LIN {X 0,Y 150.243,Z 1030.549,A -85,B 0,C 180,E1 -31632.284,E2 -31632.284} C_VEL
LIN {X 0,Y 145.871,Z 1032.288,A -85,B 0,C 180,E1 -31632.248,E2 -31632.248} C_VEL
LIN {X 0,Y 142.516,Z 1033.901,A -85,B 0,C 180,E1 -31631.848,E2 -31631.848} C_VEL
LIN {X 0,Y 134.858,Z 1038.027,A -85,B 0,C 180,E1 -31630.012,E2 -31630.012} C_VEL
LIN {X 0,Y 127.872,Z 1041.883,A -85,B 0,C 180,E1 -31627.541,E2 -31627.541} C_VEL
LIN {X 0,Y 116.114,Z 1047.754,A -85,B 0,C 180,E1 -31622.075,E2 -31622.075} C_VEL
LIN {X 0,Y 107.865,Z 1051.272,A -85,B 0,C 180,E1 -31617.134,E2 -31617.134} C_VEL
LIN {X 0,Y 99.707,Z 1054.249,A -85,B 0,C 180,E1 -31610.636,E2 -31610.636} C_VEL
LIN {X 0,Y 93.129,Z 1056.253,A -85,B 0,C 180,E1 -31603.085,E2 -31603.085} C_VEL
LIN {X 0,Y 88.672,Z 1057.261,A -85,B 0,C 180,E1 -31594.546,E2 -31594.546} C_VEL
LIN {X 0,Y 87.304,Z 1057.479,A -85,B 0,C 180,E1 -31590,E2 -31590} C_VEL
LIN {X 0,Y 90.603,Z 1056.917,A -85,B 0,C 180,E1 -31581.075,E2 -31581.075} C_VEL
LIN {X 0,Y 96.175,Z 1055.425,A -85,B 0,C 180,E1 -31573.005,E2 -31573.005} C_VEL
LIN {X 0,Y 103.623,Z 1052.922,A -85,B 0,C 180,E1 -31565.988,E2 -31565.988} C_VEL
LIN {X 0,Y 112.387,Z 1049.426,A -85,B 0,C 180,E1 -31559.983,E2 -31559.983} C_VEL
LIN {X 0,Y 122.178,Z 1044.833,A -85,B 0,C 180,E1 -31554.886,E2 -31554.886} C_VEL
LIN {X 0,Y 132.799,Z 1039.13,A -85,B 0,C 180,E1 -31550.577,E2 -31550.577} C_VEL
LIN {X 0,Y 144.738,Z 1031.716,A -85,B 0,C 180,E1 -31546.747,E2 -31546.747} C_VEL
LIN {X 0,Y 147.093,Z 1032.029,A -85,B 0,C 180,E1 -31548.019,E2 -31548.019} C_VEL
LIN {X 0,Y 159.444,Z 1036.971,A -85,B 0,C 180,E1 -31556.874,E2 -31556.874} C_VEL
LIN {X 0,Y 170.306,Z 1040.687,A -85,B 0,C 180,E1 -31563.004,E2 -31563.004} C_VEL
LIN {X 0,Y 177.43,Z 1043.023,A -85,B 0,C 180,E1 -31566.666,E2 -31566.666} C_VEL
LIN {X 0,Y 183.591,Z 1045.123,A -85,B 0,C 180,E1 -31569.848,E2 -31569.848} C_VEL
LIN {X 0,Y 190.487,Z 1047.591,A -85,B 0,C 180,E1 -31573.587,E2 -31573.587} C_VEL
LIN {X 0,Y 195.173,Z 1049.386,A -85,B 0,C 180,E1 -31576.466,E2 -31576.466} C_VEL
LIN {X 0,Y 199.859,Z 1051.299,A -85,B 0,C 180,E1 -31579.931,E2 -31579.931} C_VEL
LIN {X 0,Y 202.169,Z 1052.273,A -85,B 0,C 180,E1 -31582.007,E2 -31582.007} C_VEL
LIN {X 0,Y 204.739,Z 1053.183,A -85,B 0,C 180,E1 -31584.534,E2 -31584.534} C_VEL
LIN {X 0,Y 205.973,Z 1053.536,A -85,B 0,C 180,E1 -31586.087,E2 -31586.087} C_VEL
LIN {X 0,Y 207.098,Z 1053.852,A -85,B 0,C 180,E1 -31588.055,E2 -31588.055} C_VEL
LIN {X 0,Y 207.701,Z 1053.995,A -85,B 0,C 180,E1 -31590,E2 -31590} C_VEL
LIN {X 0,Y 207.039,Z 1053.853,A -85,B 0,C 180,E1 -31591.945,E2 -31591.945} C_VEL
LIN {X 0,Y 205.929,Z 1053.538,A -85,B 0,C 180,E1 -31593.914,E2 -31593.914} C_VEL
LIN {X 0,Y 204.269,Z 1053.046,A -85,B 0,C 180,E1 -31595.924,E2 -31595.924} C_VEL
LIN {X 0,Y 202.172,Z 1052.273,A -85,B 0,C 180,E1 -31597.993,E2 -31597.993} C_VEL
LIN {X 0,Y 199.782,Z 1051.269,A -85,B 0,C 180,E1 -31600.13,E2 -31600.13} C_VEL
LIN {X 0,Y 195.187,Z 1049.372,A -85,B 0,C 180,E1 -31603.552,E2 -31603.552} C_VEL
LIN {X 0,Y 188.933,Z 1047.004,A -85,B 0,C 180,E1 -31607.312,E2 -31607.312} C_VEL
LIN {X 0,Y 183.594,Z 1045.123,A -85,B 0,C 180,E1 -31610.152,E2 -31610.152} C_VEL
LIN {X 0,Y 176.605,Z 1042.733,A -85,B 0,C 180,E1 -31613.756,E2 -31613.756} C_VEL
LIN {X 0,Y 167.744,Z 1039.828,A -85,B 0,C 180,E1 -31618.379,E2 -31618.379} C_VEL
LIN {X 0,Y 159.439,Z 1036.975,A -85,B 0,C 180,E1 -31623.124,E2 -31623.124} C_VEL
LIN {X 0,Y 147.046,Z 1032.03,A -85,B 0,C 180,E1 -31631.998,E2 -31631.998} C_VEL
LIN {X 0,Y 144.753,Z 1031.704,A -85,B 0,C 180,E1 -31633.26,E2 -31633.26} C_VEL
LIN {X 0,Y 132.808,Z 1039.129,A -85,B 0,C 180,E1 -31629.42,E2 -31629.42} C_VEL
LIN {X 0,Y 127.872,Z 1041.883,A -85,B 0,C 180,E1 -31627.541,E2 -31627.541} C_VEL
LIN {X 0,Y 124.316,Z 1044.033,A -85,B 0,C 180,E1 -31625.632,E2 -31625.632} C_VEL
LIN {X 0,Y 120.124,Z 1047.219,A -85,B 0,C 180,E1 -31621.692,E2 -31621.692} C_VEL
LIN {X 0,Y 117.245,Z 1049.437,A -85,B 0,C 180,E1 -31618.28,E2 -31618.28} C_VEL
LIN {X 0,Y 114.627,Z 1050.924,A -85,B 0,C 180,E1 -31615.765,E2 -31615.765} C_VEL
LIN {X 0,Y 113.568,Z 1051.363,A -85,B 0,C 180,E1 -31614.962,E2 -31614.962} C_VEL
LIN {X 0,Y 106.502,Z 1054.042,A -85,B 0,C 180,E1 -31609.265,E2 -31609.265} C_VEL
LIN {X 0,Y 100.17,Z 1056.048,A -85,B 0,C 180,E1 -31602.15,E2 -31602.15} C_VEL
LIN {X 0,Y 95.82,Z 1057.056,A -85,B 0,C 180,E1 -31594.206,E2 -31594.206} C_VEL
LIN {X 0,Y 94.487,Z 1057.271,A -85,B 0,C 180,E1 -31590,E2 -31590} C_VEL
LIN {X 0,Y 97.723,Z 1056.707,A -85,B 0,C 180,E1 -31581.73,E2 -31581.73} C_VEL
LIN {X 0,Y 103.105,Z 1055.215,A -85,B 0,C 180,E1 -31574.178,E2 -31574.178} C_VEL
LIN {X 0,Y 110.264,Z 1052.713,A -85,B 0,C 180,E1 -31567.516,E2 -31567.516} C_VEL
LIN {X 0,Y 121.694,Z 1047.817,A -85,B 0,C 180,E1 -31560.026,E2 -31560.026} C_VEL
LIN {X 0,Y 133.203,Z 1041.929,A -85,B 0,C 180,E1 -31554.524,E2 -31554.524} C_VEL
LIN {X 0,Y 140.572,Z 1037.625,A -85,B 0,C 180,E1 -31551.686,E2 -31551.686} C_VEL
LIN {X 0,Y 144.007,Z 1036.261,A -85,B 0,C 180,E1 -31551.337,E2 -31551.337} C_VEL
LIN {X 0,Y 155.526,Z 1040.233,A -85,B 0,C 180,E1 -31559.156,E2 -31559.156} C_VEL
LIN {X 0,Y 166.011,Z 1043.383,A -85,B 0,C 180,E1 -31564.955,E2 -31564.955} C_VEL
LIN {X 0,Y 173.411,Z 1045.582,A -85,B 0,C 180,E1 -31568.769,E2 -31568.769} C_VEL
LIN {X 0,Y 179.086,Z 1047.306,A -85,B 0,C 180,E1 -31571.703,E2 -31571.703} C_VEL
LIN {X 0,Y 184.227,Z 1048.943,A -85,B 0,C 180,E1 -31574.512,E2 -31574.512} C_VEL
LIN {X 0,Y 188.349,Z 1050.345,A -85,B 0,C 180,E1 -31577.063,E2 -31577.063} C_VEL
LIN {X 0,Y 192.586,Z 1051.852,A -85,B 0,C 180,E1 -31580.16,E2 -31580.16} C_VEL
LIN {X 0,Y 194.344,Z 1052.503,A -85,B 0,C 180,E1 -31581.683,E2 -31581.683} C_VEL
LIN {X 0,Y 197.604,Z 1053.499,A -85,B 0,C 180,E1 -31584.766,E2 -31584.766} C_VEL
LIN {X 0,Y 198.569,Z 1053.753,A -85,B 0,C 180,E1 -31585.941,E2 -31585.941} C_VEL
LIN {X 0,Y 199.858,Z 1054.061,A -85,B 0,C 180,E1 -31587.985,E2 -31587.985} C_VEL
LIN {X 0,Y 200.561,Z 1054.201,A -85,B 0,C 180,E1 -31590,E2 -31590} C_VEL
LIN {X 0,Y 199.804,Z 1054.063,A -85,B 0,C 180,E1 -31592.016,E2 -31592.016} C_VEL
LIN {X 0,Y 198.542,Z 1053.754,A -85,B 0,C 180,E1 -31594.06,E2 -31594.06} C_VEL
LIN {X 0,Y 196.641,Z 1053.266,A -85,B 0,C 180,E1 -31596.155,E2 -31596.155} C_VEL
LIN {X 0,Y 194.346,Z 1052.503,A -85,B 0,C 180,E1 -31598.317,E2 -31598.317} C_VEL
LIN {X 0,Y 191.609,Z 1051.509,A -85,B 0,C 180,E1 -31600.567,E2 -31600.567} C_VEL
LIN {X 0,Y 187.779,Z 1050.123,A -85,B 0,C 180,E1 -31603.324,E2 -31603.324} C_VEL
LIN {X 0,Y 182.974,Z 1048.542,A -85,B 0,C 180,E1 -31606.213,E2 -31606.213} C_VEL
LIN {X 0,Y 178.16,Z 1047.031,A -85,B 0,C 180,E1 -31608.786,E2 -31608.786} C_VEL
LIN {X 0,Y 172.988,Z 1045.453,A -85,B 0,C 180,E1 -31611.447,E2 -31611.447} C_VEL
LIN {X 0,Y 164.203,Z 1042.821,A -85,B 0,C 180,E1 -31615.999,E2 -31615.999} C_VEL
LIN {X 0,Y 155.525,Z 1040.234,A -85,B 0,C 180,E1 -31620.843,E2 -31620.843} C_VEL
LIN {X 0,Y 143.975,Z 1036.285,A -85,B 0,C 180,E1 -31628.647,E2 -31628.647} C_VEL
LIN {X 0,Y 140.562,Z 1037.636,A -85,B 0,C 180,E1 -31628.304,E2 -31628.304} C_VEL
LIN {X 0,Y 130.674,Z 1043.278,A -85,B 0,C 180,E1 -31624.382,E2 -31624.382} C_VEL
LIN {X 0,Y 121.635,Z 1047.853,A -85,B 0,C 180,E1 -31619.926,E2 -31619.926} C_VEL
LIN {X 0,Y 113.568,Z 1051.363,A -85,B 0,C 180,E1 -31614.962,E2 -31614.962} C_VEL
LIN {X 0,Y 110.882,Z 1052.701,A -85,B 0,C 180,E1 -31612.353,E2 -31612.353} C_VEL
LIN {X 0,Y 108.605,Z 1054.397,A -85,B 0,C 180,E1 -31607.391,E2 -31607.391} C_VEL
LIN {X 0,Y 107.515,Z 1055.482,A -85,B 0,C 180,E1 -31603.251,E2 -31603.251} C_VEL
LIN {X 0,Y 106.317,Z 1056.086,A -85,B 0,C 180,E1 -31600.162,E2 -31600.162} C_VEL
LIN {X 0,Y 105.737,Z 1056.24,A -85,B 0,C 180,E1 -31599.148,E2 -31599.148} C_VEL
LIN {X 0,Y 101.666,Z 1057.063,A -85,B 0,C 180,E1 -31590,E2 -31590} C_VEL
LIN {X 0,Y 104.853,Z 1056.497,A -85,B 0,C 180,E1 -31582.296,E2 -31582.296} C_VEL
LIN {X 0,Y 110.069,Z 1055.005,A -85,B 0,C 180,E1 -31575.203,E2 -31575.203} C_VEL
LIN {X 0,Y 116.969,Z 1052.503,A -85,B 0,C 180,E1 -31568.869,E2 -31568.869} C_VEL
LIN {X 0,Y 127.389,Z 1047.901,A -85,B 0,C 180,E1 -31561.969,E2 -31561.969} C_VEL
LIN {X 0,Y 136.655,Z 1043.072,A -85,B 0,C 180,E1 -31557.317,E2 -31557.317} C_VEL
LIN {X 0,Y 139.142,Z 1041.722,A -85,B 0,C 180,E1 -31556.249,E2 -31556.249} C_VEL
LIN {X 0,Y 142.39,Z 1040.451,A -85,B 0,C 180,E1 -31555.667,E2 -31555.667} C_VEL
LIN {X 0,Y 153.919,Z 1043.77,A -85,B 0,C 180,E1 -31562.833,E2 -31562.833} C_VEL
LIN {X 0,Y 161.691,Z 1045.808,A -85,B 0,C 180,E1 -31566.972,E2 -31566.972} C_VEL
LIN {X 0,Y 170.451,Z 1048.132,A -85,B 0,C 180,E1 -31571.498,E2 -31571.498} C_VEL
LIN {X 0,Y 175.375,Z 1049.468,A -85,B 0,C 180,E1 -31574.104,E2 -31574.104} C_VEL
LIN {X 0,Y 180.338,Z 1050.909,A -85,B 0,C 180,E1 -31576.973,E2 -31576.973} C_VEL
LIN {X 0,Y 185.314,Z 1052.397,A -85,B 0,C 180,E1 -31580.411,E2 -31580.411} C_VEL
LIN {X 0,Y 188.921,Z 1053.487,A -85,B 0,C 180,E1 -31583.593,E2 -31583.593} C_VEL
LIN {X 0,Y 191.147,Z 1053.97,A -85,B 0,C 180,E1 -31585.783,E2 -31585.783} C_VEL
LIN {X 0,Y 192.591,Z 1054.272,A -85,B 0,C 180,E1 -31587.909,E2 -31587.909} C_VEL
LIN {X 0,Y 193.41,Z 1054.408,A -85,B 0,C 180,E1 -31590,E2 -31590} C_VEL
LIN {X 0,Y 192.547,Z 1054.273,A -85,B 0,C 180,E1 -31592.092,E2 -31592.092} C_VEL
LIN {X 0,Y 190.466,Z 1053.818,A -85,B 0,C 180,E1 -31594.959,E2 -31594.959} C_VEL
LIN {X 0,Y 186.463,Z 1052.735,A -85,B 0,C 180,E1 -31598.671,E2 -31598.671} C_VEL
LIN {X 0,Y 183.272,Z 1051.754,A -85,B 0,C 180,E1 -31601.054,E2 -31601.054} C_VEL
LIN {X 0,Y 179.422,Z 1050.611,A -85,B 0,C 180,E1 -31603.592,E2 -31603.592} C_VEL
LIN {X 0,Y 174.554,Z 1049.23,A -85,B 0,C 180,E1 -31606.369,E2 -31606.369} C_VEL
LIN {X 0,Y 168.579,Z 1047.629,A -85,B 0,C 180,E1 -31609.482,E2 -31609.482} C_VEL
LIN {X 0,Y 160.872,Z 1045.593,A -85,B 0,C 180,E1 -31613.45,E2 -31613.45} C_VEL
LIN {X 0,Y 151.771,Z 1043.164,A -85,B 0,C 180,E1 -31618.381,E2 -31618.381} C_VEL
LIN {X 0,Y 142.355,Z 1040.48,A -85,B 0,C 180,E1 -31624.31,E2 -31624.31} C_VEL
LIN {X 0,Y 139.148,Z 1041.722,A -85,B 0,C 180,E1 -31623.75,E2 -31623.75} C_VEL
LIN {X 0,Y 129.569,Z 1046.846,A -85,B 0,C 180,E1 -31619.22,E2 -31619.22} C_VEL
LIN {X 0,Y 120.873,Z 1050.86,A -85,B 0,C 180,E1 -31614.016,E2 -31614.016} C_VEL
LIN {X 0,Y 113.332,Z 1053.835,A -85,B 0,C 180,E1 -31608.062,E2 -31608.062} C_VEL
LIN {X 0,Y 107.225,Z 1055.842,A -85,B 0,C 180,E1 -31601.34,E2 -31601.34} C_VEL
LIN {X 0,Y 105.737,Z 1056.24,A -85,B 0,C 180,E1 -31599.148,E2 -31599.148} C_VEL
LIN {X 0,Y 104.785,Z 1056.693,A -85,B 0,C 180,E1 -31595.98,E2 -31595.98} C_VEL
LIN {X 0,Y 105.407,Z 1056.927,A -85,B 0,C 180,E1 -31592.747,E2 -31592.747} C_VEL
LIN {X 0,Y 110.752,Z 1056.579,A -85,B 0,C 180,E1 -31584.607,E2 -31584.607} C_VEL
LIN {X 0,Y 112.081,Z 1056.258,A -85,B 0,C 180,E1 -31582.633,E2 -31582.633} C_VEL
LIN {X 0,Y 117.037,Z 1054.795,A -85,B 0,C 180,E1 -31576.102,E2 -31576.102} C_VEL
LIN {X 0,Y 123.731,Z 1052.294,A -85,B 0,C 180,E1 -31570.075,E2 -31570.075} C_VEL
LIN {X 0,Y 133.202,Z 1047.997,A -85,B 0,C 180,E1 -31563.758,E2 -31563.758} C_VEL
LIN {X 0,Y 140.434,Z 1044.211,A -85,B 0,C 180,E1 -31559.971,E2 -31559.971} C_VEL
LIN {X 0,Y 141.344,Z 1044.181,A -85,B 0,C 180,E1 -31560.184,E2 -31560.184} C_VEL
LIN {X 0,Y 152.934,Z 1046.976,A -85,B 0,C 180,E1 -31566.79,E2 -31566.79} C_VEL
LIN {X 0,Y 157.777,Z 1048.079,A -85,B 0,C 180,E1 -31569.293,E2 -31569.293} C_VEL
LIN {X 0,Y 164.224,Z 1049.538,A -85,B 0,C 180,E1 -31572.569,E2 -31572.569} C_VEL
LIN {X 0,Y 169.965,Z 1050.893,A -85,B 0,C 180,E1 -31575.635,E2 -31575.635} C_VEL
LIN {X 0,Y 174.624,Z 1052.008,A -85,B 0,C 180,E1 -31578.391,E2 -31578.391} C_VEL
LIN {X 0,Y 178.327,Z 1052.975,A -85,B 0,C 180,E1 -31580.93,E2 -31580.93} C_VEL
LIN {X 0,Y 181.132,Z 1053.71,A -85,B 0,C 180,E1 -31583.316,E2 -31583.316} C_VEL
LIN {X 0,Y 183.633,Z 1054.189,A -85,B 0,C 180,E1 -31585.61,E2 -31585.61} C_VEL
LIN {X 0,Y 185.268,Z 1054.484,A -85,B 0,C 180,E1 -31587.826,E2 -31587.826} C_VEL
LIN {X 0,Y 186.245,Z 1054.615,A -85,B 0,C 180,E1 -31590,E2 -31590} C_VEL
LIN {X 0,Y 185.234,Z 1054.485,A -85,B 0,C 180,E1 -31592.174,E2 -31592.174} C_VEL
LIN {X 0,Y 183.327,Z 1054.142,A -85,B 0,C 180,E1 -31594.647,E2 -31594.647} C_VEL
LIN {X 0,Y 181.133,Z 1053.71,A -85,B 0,C 180,E1 -31596.684,E2 -31596.684} C_VEL
LIN {X 0,Y 178.03,Z 1052.911,A -85,B 0,C 180,E1 -31599.285,E2 -31599.285} C_VEL
LIN {X 0,Y 172.903,Z 1051.58,A -85,B 0,C 180,E1 -31602.705,E2 -31602.705} C_VEL
LIN {X 0,Y 167.791,Z 1050.348,A -85,B 0,C 180,E1 -31605.561,E2 -31605.561} C_VEL
LIN {X 0,Y 162.755,Z 1049.213,A -85,B 0,C 180,E1 -31608.199,E2 -31608.199} C_VEL
LIN {X 0,Y 157.365,Z 1047.978,A -85,B 0,C 180,E1 -31610.933,E2 -31610.933} C_VEL
LIN {X 0,Y 148.257,Z 1045.871,A -85,B 0,C 180,E1 -31615.755,E2 -31615.755} C_VEL
LIN {X 0,Y 141.28,Z 1044.183,A -85,B 0,C 180,E1 -31619.831,E2 -31619.831} C_VEL
LIN {X 0,Y 140.446,Z 1044.211,A -85,B 0,C 180,E1 -31620.026,E2 -31620.026} C_VEL
LIN {X 0,Y 131.596,Z 1048.794,A -85,B 0,C 180,E1 -31615.292,E2 -31615.292} C_VEL
LIN {X 0,Y 123.731,Z 1052.294,A -85,B 0,C 180,E1 -31609.925,E2 -31609.925} C_VEL
LIN {X 0,Y 117.069,Z 1054.794,A -85,B 0,C 180,E1 -31603.894,E2 -31603.894} C_VEL
LIN {X 0,Y 111.993,Z 1056.287,A -85,B 0,C 180,E1 -31597.21,E2 -31597.21} C_VEL
LIN {X 0,Y 108.843,Z 1056.855,A -85,B 0,C 180,E1 -31590,E2 -31590} C_VEL
LIN {X 0,Y 112.081,Z 1056.258,A -85,B 0,C 180,E1 -31582.633,E2 -31582.633} C_VEL
LIN {X 0,Y 114.591,Z 1055.735,A -85,B 0,C 180,E1 -31579.944,E2 -31579.944} C_VEL
LIN {X 0,Y 120.849,Z 1054.605,A -85,B 0,C 180,E1 -31576.233,E2 -31576.233} C_VEL
LIN {X 0,Y 126.297,Z 1053.444,A -85,B 0,C 180,E1 -31573.599,E2 -31573.599} C_VEL
LIN {X 0,Y 129.913,Z 1052.334,A -85,B 0,C 180,E1 -31571.564,E2 -31571.564} C_VEL
LIN {X 0,Y 130.932,Z 1051.9,A -85,B 0,C 180,E1 -31570.846,E2 -31570.846} C_VEL
LIN {X 0,Y 139.115,Z 1048.106,A -85,B 0,C 180,E1 -31565.412,E2 -31565.412} C_VEL
LIN {X 0,Y 141.408,Z 1047.547,A -85,B 0,C 180,E1 -31565.095,E2 -31565.095} C_VEL
LIN {X 0,Y 149.912,Z 1049.284,A -85,B 0,C 180,E1 -31569.652,E2 -31569.652} C_VEL
LIN {X 0,Y 154.983,Z 1050.24,A -85,B 0,C 180,E1 -31572.225,E2 -31572.225} C_VEL
LIN {X 0,Y 160.163,Z 1051.267,A -85,B 0,C 180,E1 -31574.873,E2 -31574.873} C_VEL
LIN {X 0,Y 165.455,Z 1052.279,A -85,B 0,C 180,E1 -31577.738,E2 -31577.738} C_VEL
LIN {X 0,Y 170.723,Z 1053.401,A -85,B 0,C 180,E1 -31581.102,E2 -31581.102} C_VEL
LIN {X 0,Y 173.168,Z 1053.939,A -85,B 0,C 180,E1 -31583.007,E2 -31583.007} C_VEL
LIN {X 0,Y 176.195,Z 1054.464,A -85,B 0,C 180,E1 -31585.689,E2 -31585.689} C_VEL
LIN {X 0,Y 177.906,Z 1054.697,A -85,B 0,C 180,E1 -31587.736,E2 -31587.736} C_VEL
LIN {X 0,Y 179.056,Z 1054.823,A -85,B 0,C 180,E1 -31590,E2 -31590} C_VEL
LIN {X 0,Y 177.883,Z 1054.698,A -85,B 0,C 180,E1 -31592.264,E2 -31592.264} C_VEL
LIN {X 0,Y 175.896,Z 1054.415,A -85,B 0,C 180,E1 -31594.583,E2 -31594.583} C_VEL
LIN {X 0,Y 173.174,Z 1053.939,A -85,B 0,C 180,E1 -31596.993,E2 -31596.993} C_VEL
LIN {X 0,Y 169.794,Z 1053.227,A -85,B 0,C 180,E1 -31599.53,E2 -31599.53} C_VEL
LIN {X 0,Y 165.435,Z 1052.265,A -85,B 0,C 180,E1 -31602.295,E2 -31602.295} C_VEL
LIN {X 0,Y 159.873,Z 1051.196,A -85,B 0,C 180,E1 -31605.293,E2 -31605.293} C_VEL
LIN {X 0,Y 153.08,Z 1049.873,A -85,B 0,C 180,E1 -31608.746,E2 -31608.746} C_VEL
LIN {X 0,Y 142.601,Z 1047.794,A -85,B 0,C 180,E1 -31614.253,E2 -31614.253} C_VEL
LIN {X 0,Y 141.407,Z 1047.548,A -85,B 0,C 180,E1 -31614.904,E2 -31614.904} C_VEL
LIN {X 0,Y 139.085,Z 1048.128,A -85,B 0,C 180,E1 -31614.561,E2 -31614.561} C_VEL
LIN {X 0,Y 130.532,Z 1052.085,A -85,B 0,C 180,E1 -31608.847,E2 -31608.847} C_VEL
LIN {X 0,Y 124.077,Z 1054.584,A -85,B 0,C 180,E1 -31603.095,E2 -31603.095} C_VEL
LIN {X 0,Y 119.125,Z 1056.078,A -85,B 0,C 180,E1 -31596.776,E2 -31596.776} C_VEL
LIN {X 0,Y 116.023,Z 1056.648,A -85,B 0,C 180,E1 -31590,E2 -31590} C_VEL
LIN {X 0,Y 119.119,Z 1056.078,A -85,B 0,C 180,E1 -31583.224,E2 -31583.224} C_VEL
LIN {X 0,Y 124.052,Z 1054.585,A -85,B 0,C 180,E1 -31576.903,E2 -31576.903} C_VEL
LIN {X 0,Y 130.932,Z 1051.9,A -85,B 0,C 180,E1 -31570.846,E2 -31570.846} C_VEL
LIN {X 0,Y 132.37,Z 1051.535,A -85,B 0,C 180,E1 -31570.358,E2 -31570.358} C_VEL
LIN {X 0,Y 135.523,Z 1051.163,A -85,B 0,C 180,E1 -31570.252,E2 -31570.252} C_VEL
LIN {X 0,Y 138.514,Z 1051.045,A -85,B 0,C 180,E1 -31570.633,E2 -31570.633} C_VEL
LIN {X 0,Y 142.602,Z 1051.118,A -85,B 0,C 180,E1 -31571.606,E2 -31571.606} C_VEL
LIN {X 0,Y 146.983,Z 1051.519,A -85,B 0,C 180,E1 -31573.202,E2 -31573.202} C_VEL
LIN {X 0,Y 150.418,Z 1051.934,A -85,B 0,C 180,E1 -31574.603,E2 -31574.603} C_VEL
LIN {X 0,Y 155.131,Z 1052.538,A -85,B 0,C 180,E1 -31576.789,E2 -31576.789} C_VEL
LIN {X 0,Y 156.572,Z 1052.762,A -85,B 0,C 180,E1 -31577.538,E2 -31577.538} C_VEL
LIN {X 0,Y 160.822,Z 1053.492,A -85,B 0,C 180,E1 -31579.933,E2 -31579.933} C_VEL
LIN {X 0,Y 163.424,Z 1053.892,A -85,B 0,C 180,E1 -31581.529,E2 -31581.529} C_VEL
LIN {X 0,Y 164.978,Z 1054.174,A -85,B 0,C 180,E1 -31582.658,E2 -31582.658} C_VEL
LIN {X 0,Y 169.067,Z 1054.79,A -85,B 0,C 180,E1 -31586.067,E2 -31586.067} C_VEL
LIN {X 0,Y 170.436,Z 1054.913,A -85,B 0,C 180,E1 -31587.637,E2 -31587.637} C_VEL
LIN {X 0,Y 171.838,Z 1055.032,A -85,B 0,C 180,E1 -31590,E2 -31590} C_VEL
LIN {X 0,Y 170.421,Z 1054.914,A -85,B 0,C 180,E1 -31592.363,E2 -31592.363} C_VEL
LIN {X 0,Y 169.067,Z 1054.79,A -85,B 0,C 180,E1 -31593.933,E2 -31593.933} C_VEL
LIN {X 0,Y 164.985,Z 1054.174,A -85,B 0,C 180,E1 -31597.342,E2 -31597.342} C_VEL
LIN {X 0,Y 163.426,Z 1053.89,A -85,B 0,C 180,E1 -31598.476,E2 -31598.476} C_VEL
LIN {X 0,Y 157.93,Z 1052.981,A -85,B 0,C 180,E1 -31601.764,E2 -31601.764} C_VEL
LIN {X 0,Y 152.521,Z 1052.109,A -85,B 0,C 180,E1 -31604.617,E2 -31604.617} C_VEL
LIN {X 0,Y 147.225,Z 1051.228,A -85,B 0,C 180,E1 -31607.31,E2 -31607.31} C_VEL
LIN {X 0,Y 140.927,Z 1050.242,A -85,B 0,C 180,E1 -31610.431,E2 -31610.431} C_VEL
LIN {X 0,Y 134.083,Z 1053.212,A -85,B 0,C 180,E1 -31605.193,E2 -31605.193} C_VEL
LIN {X 0,Y 128.046,Z 1055.357,A -85,B 0,C 180,E1 -31598.909,E2 -31598.909} C_VEL
LIN {X 0,Y 124.481,Z 1056.234,A -85,B 0,C 180,E1 -31593.236,E2 -31593.236} C_VEL
LIN {X 0,Y 123.204,Z 1056.44,A -85,B 0,C 180,E1 -31590,E2 -31590} C_VEL
LIN {X 0,Y 126.252,Z 1055.869,A -85,B 0,C 180,E1 -31583.608,E2 -31583.608} C_VEL
LIN {X 0,Y 131.089,Z 1054.375,A -85,B 0,C 180,E1 -31577.617,E2 -31577.617} C_VEL
LIN {X 0,Y 137.368,Z 1051.876,A -85,B 0,C 180,E1 -31572.124,E2 -31572.124} C_VEL
LIN {X 0,Y 141.069,Z 1050.237,A -85,B 0,C 180,E1 -31569.591,E2 -31569.591} C_VEL
LIN {X 0,Y 148.923,Z 1051.526,A -85,B 0,C 180,E1 -31573.552,E2 -31573.552} C_VEL
LIN {X 0,Y 155.469,Z 1052.575,A -85,B 0,C 180,E1 -31576.937,E2 -31576.937} C_VEL
LIN {X 0,Y 156.572,Z 1052.762,A -85,B 0,C 180,E1 -31577.538,E2 -31577.538} C_VEL
LIN {X 0,Y 158.464,Z 1053.187,A -85,B 0,C 180,E1 -31578.787,E2 -31578.787} C_VEL
LIN {X 0,Y 160.315,Z 1053.815,A -85,B 0,C 180,E1 -31580.802,E2 -31580.802} C_VEL
LIN {X 0,Y 161.368,Z 1054.385,A -85,B 0,C 180,E1 -31582.891,E2 -31582.891} C_VEL
LIN {X 0,Y 163.626,Z 1055.181,A -85,B 0,C 180,E1 -31588.644,E2 -31588.644} C_VEL
LIN {X 0,Y 164.577,Z 1055.243,A -85,B 0,C 180,E1 -31590,E2 -31590} C_VEL
LIN {X 0,Y 162.913,Z 1055.131,A -85,B 0,C 180,E1 -31592.472,E2 -31592.472} C_VEL
LIN {X 0,Y 160.006,Z 1054.88,A -85,B 0,C 180,E1 -31595.04,E2 -31595.04} C_VEL
LIN {X 0,Y 156.106,Z 1054.386,A -85,B 0,C 180,E1 -31597.93,E2 -31597.93} C_VEL
LIN {X 0,Y 150.437,Z 1053.676,A -85,B 0,C 180,E1 -31601.174,E2 -31601.174} C_VEL
LIN {X 0,Y 143.3,Z 1052.69,A -85,B 0,C 180,E1 -31604.811,E2 -31604.811} C_VEL
LIN {X 0,Y 141.052,Z 1053.003,A -85,B 0,C 180,E1 -31604.426,E2 -31604.426} C_VEL
LIN {X 0,Y 134.866,Z 1055.245,A -85,B 0,C 180,E1 -31598.073,E2 -31598.073} C_VEL
LIN {X 0,Y 130.384,Z 1056.232,A -85,B 0,C 180,E1 -31590,E2 -31590} C_VEL
LIN {X 0,Y 134.866,Z 1055.244,A -85,B 0,C 180,E1 -31581.925,E2 -31581.925} C_VEL
LIN {X 0,Y 141.044,Z 1053.003,A -85,B 0,C 180,E1 -31575.574,E2 -31575.574} C_VEL
LIN {X 0,Y 143.296,Z 1052.69,A -85,B 0,C 180,E1 -31575.187,E2 -31575.187} C_VEL
LIN {X 0,Y 151.28,Z 1053.775,A -85,B 0,C 180,E1 -31579.291,E2 -31579.291} C_VEL
LIN {X 0,Y 156.403,Z 1054.421,A -85,B 0,C 180,E1 -31582.253,E2 -31582.253} C_VEL
LIN {X 0,Y 160.002,Z 1054.88,A -85,B 0,C 180,E1 -31584.96,E2 -31584.96} C_VEL
LIN {X 0,Y 162.92,Z 1055.131,A -85,B 0,C 180,E1 -31587.528,E2 -31587.528} C_VEL
LIN {X 0,Y 163.626,Z 1055.181,A -85,B 0,C 180,E1 -31588.644,E2 -31588.644} C_VEL
LIN {X 0,Y 163.6,Z 1055.244,A -85,B 0,C 180,E1 -31589.51,E2 -31589.51} C_VEL
LIN {X 0,Y 162.056,Z 1055.288,A -85,B 0,C 180,E1 -31590.743,E2 -31590.743} C_VEL
LIN {X 0,Y 159.552,Z 1055.282,A -85,B 0,C 180,E1 -31591.841,E2 -31591.841} C_VEL
LIN {X 0,Y 153.045,Z 1055.247,A -85,B 0,C 180,E1 -31594.409,E2 -31594.409} C_VEL
LIN {X 0,Y 151.956,Z 1055.14,A -85,B 0,C 180,E1 -31595.122,E2 -31595.122} C_VEL
LIN {X 0,Y 148.777,Z 1054.859,A -85,B 0,C 180,E1 -31597.258,E2 -31597.258} C_VEL
LIN {X 0,Y 145.241,Z 1054.498,A -85,B 0,C 180,E1 -31599.302,E2 -31599.302} C_VEL
LIN {X 0,Y 142.706,Z 1054.816,A -85,B 0,C 180,E1 -31598.496,E2 -31598.496} C_VEL
LIN {X 0,Y 138.849,Z 1055.823,A -85,B 0,C 180,E1 -31592.901,E2 -31592.901} C_VEL
LIN {X 0,Y 137.557,Z 1056.024,A -85,B 0,C 180,E1 -31590,E2 -31590} C_VEL
LIN {X 0,Y 141.703,Z 1055.138,A -85,B 0,C 180,E1 -31582.709,E2 -31582.709} C_VEL
LIN {X 0,Y 142.702,Z 1054.816,A -85,B 0,C 180,E1 -31581.504,E2 -31581.504} C_VEL
LIN {X 0,Y 145.221,Z 1054.501,A -85,B 0,C 180,E1 -31580.705,E2 -31580.705} C_VEL
LIN {X 0,Y 148.774,Z 1054.861,A -85,B 0,C 180,E1 -31582.753,E2 -31582.753} C_VEL
LIN {X 0,Y 151.704,Z 1055.123,A -85,B 0,C 180,E1 -31584.684,E2 -31584.684} C_VEL
LIN {X 0,Y 155.261,Z 1055.353,A -85,B 0,C 180,E1 -31587.406,E2 -31587.406} C_VEL
LIN {X 0,Y 157.271,Z 1055.454,A -85,B 0,C 180,E1 -31590,E2 -31590} C_VEL
LIN {X 0,Y 154.818,Z 1055.336,A -85,B 0,C 180,E1 -31592.951,E2 -31592.951} C_VEL
LIN {X 0,Y 151.956,Z 1055.14,A -85,B 0,C 180,E1 -31595.122,E2 -31595.122} C_VEL
LIN {X 0,Y 150.878,Z 1055.18,A -85,B 0,C 180,E1 -31595.217,E2 -31595.217} C_VEL
LIN {X 0,Y 148.63,Z 1055.377,A -85,B 0,C 180,E1 -31594.571,E2 -31594.571} C_VEL
LIN {X 0,Y 146.469,Z 1055.593,A -85,B 0,C 180,E1 -31592.922,E2 -31592.922} C_VEL
LIN {X 0,Y 145.339,Z 1055.717,A -85,B 0,C 180,E1 -31591.381,E2 -31591.381} C_VEL
LIN {X 0,Y 144.726,Z 1055.817,A -85,B 0,C 180,E1 -31590,E2 -31590} C_VEL
LIN {X 0,Y 146.023,Z 1055.617,A -85,B 0,C 180,E1 -31587.241,E2 -31587.241} C_VEL
LIN {X 0,Y 147.122,Z 1055.586,A -85,B 0,C 180,E1 -31587.262,E2 -31587.262} C_VEL
LIN {X 0,Y 149.854,Z 1055.669,A -85,B 0,C 180,E1 -31590,E2 -31590} C_VEL
LIN {X 0,Y 147.127,Z 1055.586,A -85,B 0,C 180,E1 -31592.738,E2 -31592.738} C_VEL
LIN {X 0,Y 146.04,Z 1055.617,A -85,B 0,C 180,E1 -31592.758,E2 -31592.758} C_VEL
LIN {X 0,Y 145.339,Z 1055.717,A -85,B 0,C 180,E1 -31591.381,E2 -31591.381} C_VEL
LIN {X 0,Y 145.339,Z 1055.717,A -85,B 0,C 180,E1 -31591.381,E2 -31591.381}

QRS_NEXT_CUT()

QRS_NEXT()
QRS_HOME()

END
